PROGRAM Auto_Manual
VAR
END_VAR

IF gvl.ixAuto THEN
	Auto_Mode();	
END_IF

END_PROGRAM

(* stored: Version 1.1.0.1, ProductVersion 3.1.4024.12
   POU Auto_Manual: Id {c8ad19c2-a76a-4b26-9eca-0b80aee427ec}, SpecialFunc None *)
